// TIA Portal V16 export
// export: Created 2021-07-12T14:47:17.7455569Z, ExportSetting WithDefaults, DisplayName Totally Integrated Automation Portal, DisplayVersion V16, DisplayName TIA Portal Version Control Interface, DisplayVersion V16, DisplayName TIA Portal Openness, DisplayVersion V16, DisplayName STEP 7 Professional, DisplayVersion V16, DisplayName STEP 7 Safety, DisplayVersion V16, DisplayName WinCC Professional, DisplayVersion V16
TYPE "LSimaHydTO_typeInternalControl"
TITLE = LSimaHydTO_typeInternalControl
// Command structure, use for axis control
// stored: IsFailsafeCompliant false
   STRUCT
      AckError : Bool;   // Acknowledge error of axis
      ExecuteForceLimiting : Bool;   // Rising edge starts force limiting defined by ForceCommand
      ExecuteForceControl : Bool;   // Rising edge starts force control defined by ForceCommand
      RequestForward : Bool;   // request to open direction valve forward
      RequestBackward : Bool;   // request to open direction valve backward
      ForceCommand { S7_SetPoint := 'True'} : "LSimaHydTO_typeInternalControlForceCmd";   // Defines force command
      DirectOutput { S7_SetPoint := 'True'} : "LSimaHydTO_typeInternalControlDirectOutput";
   END_STRUCT;
END_TYPE
